FUNCTION_BLOCK A2X_XOR_2 (* Composite FB to calculate boolean XOR between 2 A2X adapters (UP and DOWN independently) *)
  (* Standard: 61499-2; Function: OUT.UP = IN1.UP XOR IN2.UP, OUT.DOWN = IN1.DOWN XOR IN2.DOWN; Description: Copyright (c) 2026 HR Agrartechnik GmbH This program and the accompanying materials are made available under the terms of the Eclipse Public License 2.0 which is available at https://www.eclipse.org/legal/epl-2.0/ SPDX-License-Identifier: EPL-2.0 *)
  (* Version 1.0, 2026-08-31, Franz Höpfinger, HR Agrartechnik GmbH, Initial Version *)
  PACKAGE adapter::booleanOperators;
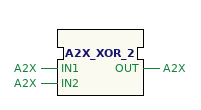
  SOCKETS
    IN1 : adapter::types::unidirectional::A2X; (* XOR input 1 *)
    IN2 : adapter::types::unidirectional::A2X; (* XOR input 2 *)
  END_SOCKETS
  PLUGS
    OUT : adapter::types::unidirectional::A2X; (* XOR result *)
  END_PLUGS
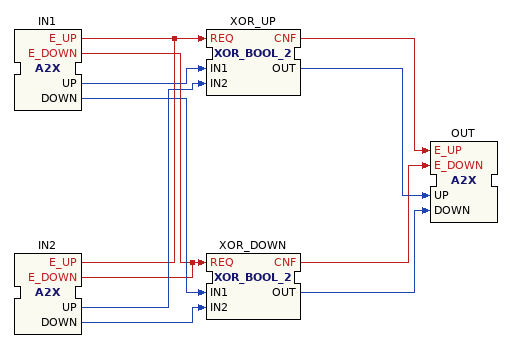
  FBS
    XOR_UP : iec61131::booleanOperators::XOR_BOOL_2; (* XORs the UP channel *)
    XOR_DOWN : iec61131::booleanOperators::XOR_BOOL_2; (* XORs the DOWN channel *)
  END_FBS
  EVENT_CONNECTIONS
    IN1.E_UP TO XOR_UP.REQ;
    IN2.E_UP TO XOR_UP.REQ;
    XOR_UP.CNF TO OUT.E_UP;
    IN1.E_DOWN TO XOR_DOWN.REQ;
    IN2.E_DOWN TO XOR_DOWN.REQ;
    XOR_DOWN.CNF TO OUT.E_DOWN;
  END_CONNECTIONS
  DATA_CONNECTIONS
    IN1.UP TO XOR_UP.IN1;
    IN2.UP TO XOR_UP.IN2;
    XOR_UP.OUT TO OUT.UP;
    IN1.DOWN TO XOR_DOWN.IN1;
    IN2.DOWN TO XOR_DOWN.IN2;
    XOR_DOWN.OUT TO OUT.DOWN;
  END_CONNECTIONS
END_FUNCTION_BLOCK
